FUNCTION_BLOCK FB_SVs_504_505_Ablaufsteuerung
VAR_IN_OUT
	Zustand			: ST_SVs_504_505_Zustand;
	Stellwert		: ST_SV_Stellwert;
END_VAR
VAR_INPUT
	Steuerung		: ST_SV_Steuerung;
	Parameter		: ST_SV_Parameter;
END_VAR
VAR_OUTPUT
END_VAR
VAR
	E_Stellventil_Zustand_Stellungwechsel10						: SINT;
	E_Stellventil_Zustand_Stellungwechsel01						: SINT;
	E_Stellventil_Zustand_Status_Stellungrueckmeldung0_Sperre	: SINT;
	E_Stellventil_Zustand_Status_Stellungrueckmeldung0			: SINT;
	E_Stellventil_Zustand_Status_Stellungrueckmeldung1_Sperre	: SINT;
	E_Stellventil_Zustand_Status_Stellungrueckmeldung1			: SINT;
END_VAR

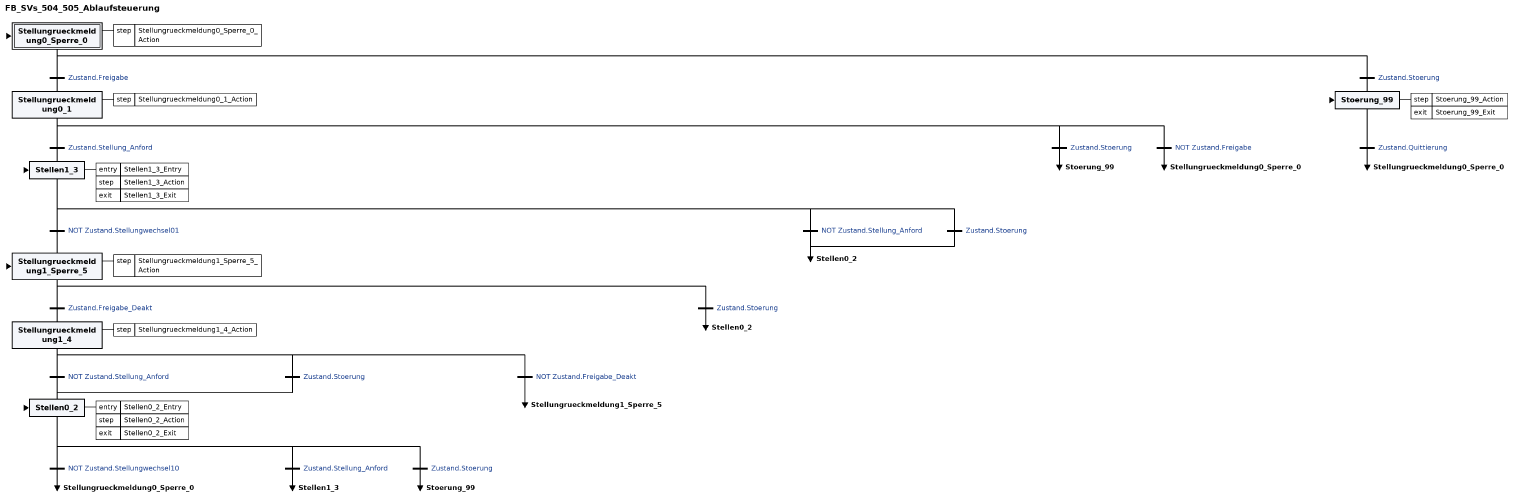
INITIAL_STEP Stellungrueckmeldung0_Sperre_0:
    Stellungrueckmeldung0_Sperre_0_Action(N);  // step action
END_STEP
TRANSITION FROM Stellungrueckmeldung0_Sperre_0 TO Stellungrueckmeldung0_1
    := Zustand.Freigabe;
END_TRANSITION
TRANSITION FROM Stellungrueckmeldung0_Sperre_0 TO Stoerung_99
    := Zustand.Stoerung;
END_TRANSITION
STEP Stoerung_99:
    Stoerung_99_Action(N);  // step action
    Stoerung_99_Exit(P0);  // exit action
END_STEP
TRANSITION FROM Stoerung_99 TO Stellungrueckmeldung0_Sperre_0
    := Zustand.Quittierung;
END_TRANSITION
STEP Stellungrueckmeldung0_1:
    Stellungrueckmeldung0_1_Action(N);  // step action
END_STEP
TRANSITION FROM Stellungrueckmeldung0_1 TO Stellen1_3
    := Zustand.Stellung_Anford;
END_TRANSITION
TRANSITION FROM Stellungrueckmeldung0_1 TO Stoerung_99
    := Zustand.Stoerung;
END_TRANSITION
TRANSITION FROM Stellungrueckmeldung0_1 TO Stellungrueckmeldung0_Sperre_0
    := NOT Zustand.Freigabe;
END_TRANSITION
STEP Stellen1_3:
    Stellen1_3_Entry(P1);  // entry action
    Stellen1_3_Action(N);  // step action
    Stellen1_3_Exit(P0);  // exit action
END_STEP
TRANSITION FROM Stellen1_3 TO Stellungrueckmeldung1_Sperre_5
    := NOT Zustand.Stellungwechsel01;
END_TRANSITION
TRANSITION FROM Stellen1_3 TO Stellen0_2
    := NOT Zustand.Stellung_Anford;
END_TRANSITION
TRANSITION FROM Stellen1_3 TO Stellen0_2
    := Zustand.Stoerung;
END_TRANSITION
STEP Stellungrueckmeldung1_Sperre_5:
    Stellungrueckmeldung1_Sperre_5_Action(N);  // step action
END_STEP
TRANSITION FROM Stellungrueckmeldung1_Sperre_5 TO Stellungrueckmeldung1_4
    := Zustand.Freigabe_Deakt;
END_TRANSITION
TRANSITION FROM Stellungrueckmeldung1_Sperre_5 TO Stellen0_2
    := Zustand.Stoerung;
END_TRANSITION
STEP Stellungrueckmeldung1_4:
    Stellungrueckmeldung1_4_Action(N);  // step action
END_STEP
TRANSITION FROM Stellungrueckmeldung1_4 TO Stellen0_2
    := NOT Zustand.Stellung_Anford;
END_TRANSITION
TRANSITION FROM Stellungrueckmeldung1_4 TO Stellen0_2
    := Zustand.Stoerung;
END_TRANSITION
TRANSITION FROM Stellungrueckmeldung1_4 TO Stellungrueckmeldung1_Sperre_5
    := NOT Zustand.Freigabe_Deakt;
END_TRANSITION
STEP Stellen0_2:
    Stellen0_2_Entry(P1);  // entry action
    Stellen0_2_Action(N);  // step action
    Stellen0_2_Exit(P0);  // exit action
END_STEP
TRANSITION FROM Stellen0_2 TO Stellungrueckmeldung0_Sperre_0
    := NOT Zustand.Stellungwechsel10;
END_TRANSITION
TRANSITION FROM Stellen0_2 TO Stellen1_3
    := Zustand.Stellung_Anford;
END_TRANSITION
TRANSITION FROM Stellen0_2 TO Stoerung_99
    := Zustand.Stoerung;
END_TRANSITION

ACTION Stellen0_2_Action:
(* Stellwert setzen *)
Stellwert.Stellung := FALSE;

(* Zustand setzen *)
Zustand.Stellungwechsel10 := NOT (Zustand.Stellungrueckmeldung0_505 AND (NOT Zustand.Stellungrueckmeldung1_505)) ;
Zustand.Status := E_Stellventil_Zustand_Stellungwechsel10;
END_ACTION

ACTION Stellen0_2_Entry:
Zustand.Stellungwechsel10 := TRUE;
END_ACTION

ACTION Stellen0_2_Exit:
Zustand.Stellungwechsel10 := FALSE;
END_ACTION

ACTION Stellen1_3_Action:
(* Stellwert setzen *)
Stellwert.Stellung := TRUE;

(* Zustand setzen *)
Zustand.Stellungwechsel01 := NOT(Zustand.Stellungrueckmeldung1_505 AND (NOT Zustand.Stellungrueckmeldung0_505));
Zustand.Status := E_Stellventil_Zustand_Stellungwechsel01;
END_ACTION

ACTION Stellen1_3_Entry:
Zustand.Stellungwechsel01 := TRUE;
END_ACTION

ACTION Stellen1_3_Exit:
Zustand.Stellungwechsel01 := FALSE;
END_ACTION

ACTION Stellungrueckmeldung0_1_Action:
(* Stellwert setzen *)
Stellwert.Stellung := FALSE;
Zustand.Stellung := FALSE;

(* Zustand setzen *)
Zustand.Status := E_Stellventil_Zustand_Status_Stellungrueckmeldung0;
END_ACTION

ACTION Stellungrueckmeldung0_Sperre_0_Action:
(* Stellwert setzen *)
Stellwert.Stellung := FALSE;
Zustand.Stellung := FALSE;

(* Zustand setzen *)
Zustand.Status := E_Stellventil_Zustand_Status_Stellungrueckmeldung0_Sperre;
END_ACTION

ACTION Stellungrueckmeldung1_4_Action:
(* Stellwert setzen *)
Stellwert.Stellung := TRUE;
Zustand.Stellung := TRUE;

(* Zustand setzen *)
Zustand.Status := E_Stellventil_Zustand_Status_Stellungrueckmeldung1;
END_ACTION

ACTION Stellungrueckmeldung1_Sperre_5_Action:
(* Stellwert setzen *)
Stellwert.Stellung := TRUE;
Zustand.Stellung := TRUE;

(* Zustand setzen *)
Zustand.Status := E_Stellventil_Zustand_Status_Stellungrueckmeldung1_Sperre;
END_ACTION

ACTION Stoerung_99_Action:
(* Stellwert setzen *)
Stellwert.Stellung := Zustand.Stellung;

(* Zustand setzen *)
Zustand.Stoerung := TRUE;
Zustand.Status := E_PU_Zustand_Status_Stoerung;
END_ACTION

ACTION Stoerung_99_Exit:
Zustand.Stoerung	:= FALSE;
END_ACTION

END_FUNCTION_BLOCK

(* stored: Version 1.1.0.1, ProductVersion 3.1.4024.9
   POU FB_SVs_504_505_Ablaufsteuerung: Id {ed4faa53-59ac-49bd-8522-5edbced3214b}, SpecialFunc None
   Action Stellen0_2_Action: Id {b7696bc9-2107-493f-a46f-26cdb5d6805d}
   Action Stellen0_2_Entry: Id {a156a96f-c647-45c2-97ef-daefce1979a5}
   Action Stellen0_2_Exit: Id {bfad2159-69ab-4a27-9913-51aebeba8969}
   Action Stellen1_3_Action: Id {249bfd4b-ed01-49ca-874b-6f1f4108dc72}
   Action Stellen1_3_Entry: Id {c3233715-5481-4131-886b-83f23e4e00f6}
   Action Stellen1_3_Exit: Id {4c5e1383-3520-4093-8b95-2857994a94c4}
   Action Stellungrueckmeldung0_1_Action: Id {406c4567-c9d6-4172-a822-f0b3488b82cb}
   Action Stellungrueckmeldung0_Sperre_0_Action: Id {403bc09c-ce51-4214-a5e2-b86ab5a7917a}
   Action Stellungrueckmeldung1_4_Action: Id {36f140ac-2d23-471d-82a6-7239a9c7bcd2}
   Action Stellungrueckmeldung1_Sperre_5_Action: Id {a3115a58-29c5-4c58-877d-844558e452bd}
   Action Stoerung_99_Action: Id {fbc829e7-1352-427f-baae-55e5dc55237c}
   Action Stoerung_99_Exit: Id {32ce2a6d-15fa-40ba-813d-99e2af3420f4} *)
